// TIA Portal V20 export
TYPE "QrReadIdVision"
// stored: Access Published, Namespace LER
   STRUCT
      Data : Struct
         QrInterfaceId : String[64];
         Vision { S7_SetPoint := 'True'} : Array[1..2] of "LER_typeVisionAlignResultData";
         Align { S7_SetPoint := 'True'} : Array[1..2] of "LER_typeVisionAlignResultData";
         verdict { S7_SetPoint := 'True'} : Array[1..2] of Bool;
      END_STRUCT;
   END_STRUCT;
END_TYPE
